{attribute 'pack_mode' := '1'}
    {attribute 'OPC.UA.DA' := '1'}
    {attribute 'OPC.UA.DA.StructuredType' := '1'}
    (*
    ST_RW_DigitalIn_HMI_IgnitionExp
    ==================================================
    Generated from Ignition UDT: RW_Digital_In
    Total tags: 7
    Generated on: 2025-09-15 12:56:43
    *)
    TYPE ST_RW_DigitalIn_HMI_IgnitionExp :
    STRUCT
        {attribute 'OPC.UA.DA' := '1'}
        Highest_Active_Property : DINT := 0;
        {attribute 'OPC.UA.DA' := '1'}
        Manual_Input : BOOL := FALSE;
        {attribute 'OPC.UA.DA' := '1'}
        AllowManualOverride : BOOL := FALSE;
        {attribute 'OPC.UA.DA' := '1'}
        Manual_Mode : BOOL := FALSE;
        {attribute 'OPC.UA.DA' := '1'}
        Input_Raw : BOOL := FALSE;

        {attribute 'OPC.UA.DA' := '1'}
        Alarm_Active : BOOL := FALSE;
        {attribute 'OPC.UA.DA' := '1'}
        Input : BOOL := FALSE;
    END_STRUCT
    END_TYPE

(* stored: Version 1.1.0.1
   DUT ST_RW_DigitalIn_HMI_IgnitionExp: Id {75b1cd9a-f182-461e-95a2-f4e31f7e43db} *)
